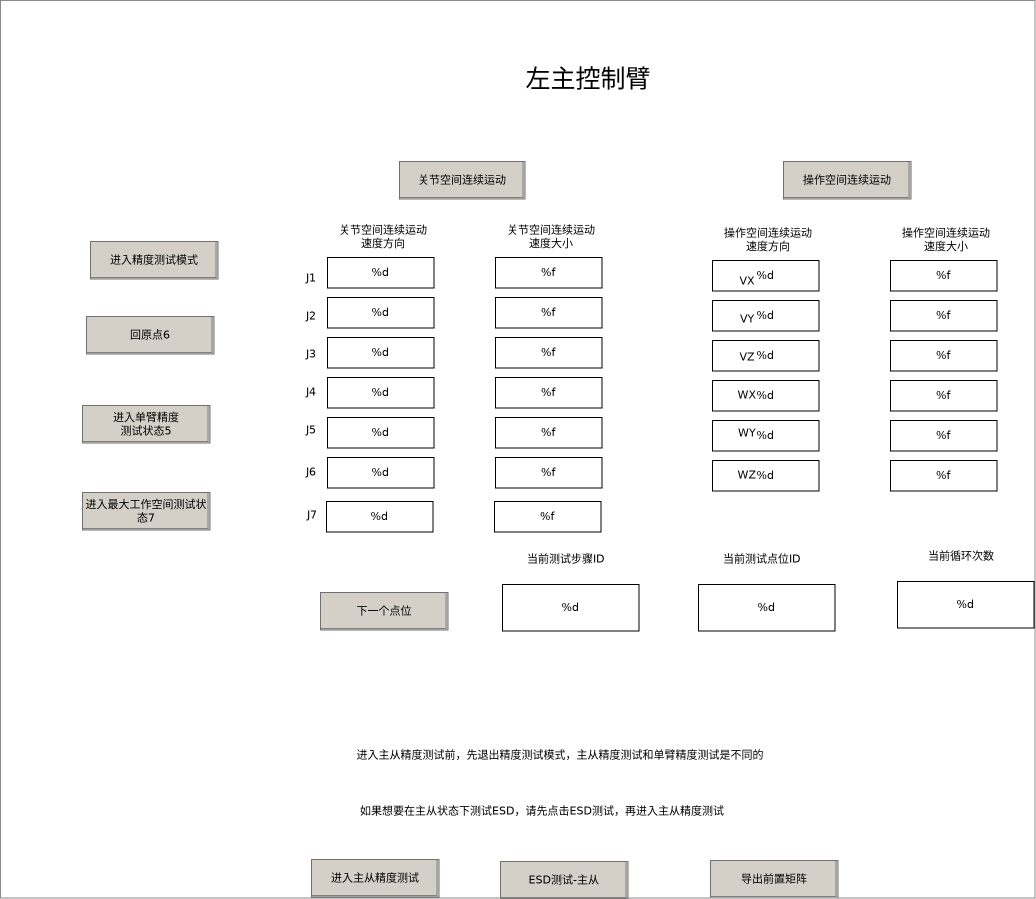
VISUALIZATION precision_a1  // 1036x899
    Label (513,57 150x43), "左主控制臂"
    Rectangle (327,257 107x31), "%d", text variable: g_motionTest.m_jntMotionDir[1][1]
        OnMouseClick: write the text variable via Default, min -1, max 1
    Label (308,222 150x29), "关节空间连续运动 速度方向"
    Rectangle (327,297 107x31), "%d", text variable: g_motionTest.m_jntMotionDir[1][2]
        OnMouseClick: write the text variable via Default, min -1, max 1
    Rectangle (327,337 107x31), "%d", text variable: g_motionTest.m_jntMotionDir[1][3]
        OnMouseClick: write the text variable via Default, min -1, max 1
    Rectangle (327,377 107x31), "%d", text variable: g_motionTest.m_jntMotionDir[1][4]
        OnMouseClick: write the text variable via Default, min -1, max 1
    Rectangle (327,417 107x31), "%d", text variable: g_motionTest.m_jntMotionDir[1][5]
        OnMouseClick: write the text variable via Default, min -1, max 1
    Rectangle (327,457 107x31), "%d", text variable: g_motionTest.m_jntMotionDir[1][6]
        OnMouseClick: write the text variable via Default, min -1, max 1
    Rectangle (495,257 107x31), "%f", text variable: g_motionTest.m_jntVel[1][1]
        OnMouseClick: write the text variable via Default
    Label (476,222 150x29), "关节空间连续运动 速度大小"
    Rectangle (495,297 107x31), "%f", text variable: g_motionTest.m_jntVel[1][2]
        OnMouseClick: write the text variable via Default
    Rectangle (495,337 107x31), "%f", text variable: g_motionTest.m_jntVel[1][3]
        OnMouseClick: write the text variable via Default
    Rectangle (495,377 107x31), "%f", text variable: g_motionTest.m_jntVel[1][4]
        OnMouseClick: write the text variable via Default
    Rectangle (495,417 107x31), "%f", text variable: g_motionTest.m_jntVel[1][5]
        OnMouseClick: write the text variable via Default
    Rectangle (495,457 107x31), "%f", text variable: g_motionTest.m_jntVel[1][6]
        OnMouseClick: write the text variable via Default
    Rectangle (712,260 107x31), "%d", text variable: g_motionTest.m_spatialMotionDir[1][1]
        OnMouseClick: write the text variable via Default, min -1, max 1
    Label (693,225 150x29), "操作空间连续运动 速度方向"
    Rectangle (712,300 107x31), "%d", text variable: g_motionTest.m_spatialMotionDir[1][2]
        OnMouseClick: write the text variable via Default, min -1, max 1
    Rectangle (712,340 107x31), "%d", text variable: g_motionTest.m_spatialMotionDir[1][3]
        OnMouseClick: write the text variable via Default, min -1, max 1
    Rectangle (712,380 107x31), "%d", text variable: g_motionTest.m_spatialMotionDir[1][4]
        OnMouseClick: write the text variable via Default, min -1, max 1
    Rectangle (712,420 107x31), "%d", text variable: g_motionTest.m_spatialMotionDir[1][5]
        OnMouseClick: write the text variable via Default, min -1, max 1
    Rectangle (712,460 107x31), "%d", text variable: g_motionTest.m_spatialMotionDir[1][6]
        OnMouseClick: write the text variable via Default, min -1, max 1
    Rectangle (890,260 107x31), "%f", text variable: g_motionTest.m_spatialVel[1][1]
        OnMouseClick: write the text variable via Default
    Label (871,225 150x29), "操作空间连续运动 速度大小"
    Rectangle (890,300 107x31), "%f", text variable: g_motionTest.m_spatialVel[1][2]
        OnMouseClick: write the text variable via Default
    Rectangle (890,340 107x31), "%f", text variable: g_motionTest.m_spatialVel[1][3]
        OnMouseClick: write the text variable via Default
    Rectangle (890,380 107x31), "%f", text variable: g_motionTest.m_spatialVel[1][4]
        OnMouseClick: write the text variable via Default
    Rectangle (890,420 107x31), "%f", text variable: g_motionTest.m_spatialVel[1][5]
        OnMouseClick: write the text variable via Default
    Rectangle (890,460 107x31), "%f", text variable: g_motionTest.m_spatialVel[1][6]
        OnMouseClick: write the text variable via Default
    Button (90,241 128x38), "进入精度测试模式", colour toggle: g_motionTest.m_enterPrecisionTestMode[1]
        toggle g_motionTest.m_enterPrecisionTestMode[1]
    Button (399,161 126x38), "关节空间连续运动", colour toggle: g_motionTest.m_uiArmModeL[1,2]
        tap g_motionTest.m_uiArmMode[1,2]
    Button (783,161 128x38), "操作空间连续运动", colour toggle: g_motionTest.m_uiArmModeL[1,4]
        tap g_motionTest.m_uiArmMode[1,4]
    Button (86,316 128x38), "回原点6", colour toggle: g_motionTest.m_uiArmModeL[1,6]
        tap g_motionTest.m_uiArmMode[1,6]
    Button (320,592 128x38), "下一个点位", colour toggle: g_motionTest.m_nextStep[1]
        tap g_motionTest.m_nextStep[1]
    Group (491,541 545x90)
        Rectangle (11,43 137x47), "%d", text variable: g_motionTest.m_curStep[1]
        Label (0,3 150x30), "当前测试步骤ID"
        Rectangle (207,43 137x47), "%d", text variable: g_motionTest.m_testPointId[1]
        Label (196,3 150x30), "当前测试点位ID"
        Rectangle (406,40 137x47), "%d", text variable: g_motionTest.m_testCycleId[1]
        Label (395,0 150x30), "当前循环次数"
    Label (304,263 14x30), "J1"
    Label (304,301 14x30), "J2"
    Label (304,339 14x30), "J3"
    Label (304,377 14x30), "J4"
    Label (304,415 14x30), "J5"
    Label (304,457 14x30), "J6"
    Group (672,266 26x224)
        Label (0,0 150x30), "VX"
        Label (0,38 150x30), "VY"
        Label (0,76 150x30), "VZ"
        Label (0,114 150x30), "WX"
        Label (0,152 150x30), "WY"
        Label (0,194 150x30), "WZ"
    Button (82,405 128x38), "进入单臂精度 测试状态5", colour toggle: g_motionTest.m_uiArmModeL[1,5]
        toggle g_motionTest.m_uiArmMode[1,5]
    Button (82,492 128x38), "进入最大工作空间测试状态7", colour toggle: g_motionTest.m_uiArmModeL[1,7]
        toggle g_motionTest.m_uiArmMode[1,7]
    Button (311,859 128x38), "进入主从精度测试", colour toggle: g_motionTest.m_MSPrecisionTest[1]
        toggle g_motionTest.m_MSPrecisionTest[1]
    Rectangle (326,501 107x31), "%d", text variable: g_motionTest.m_jntMotionDir[1][7]
        OnMouseClick: write the text variable via Default, min -1, max 1
    Rectangle (494,501 107x31), "%f", text variable: g_motionTest.m_jntVel[1][7]
        OnMouseClick: write the text variable via Default
    Label (305,500 14x30), "J7"
    Button (710,860 128x38), "导出前置矩阵"
        tap g_motionTest.m_writeData[1]
    Button (500,861 128x38), "ESD测试-主从", colour toggle: g_motionTest.m_esdTest[1]
        toggle g_motionTest.m_esdTest[1]
    Label (241,740 638x30), "进入主从精度测试前，先退出精度测试模式，主从精度测试和单臂精度测试是不同的"
    Label (223,796 638x30), "如果想要在主从状态下测试ESD，请先点击ESD测试，再进入主从精度测试"
END_VISUALIZATION

(* stored: Version 1.1.0.1, ProductVersion 3.1.4024.11
   Visu precision_a1: Id {c275d056-9c8b-436c-b15b-86e3d9a625b0} *)
